Staubli VAL3: getFullError.pgx

public program getFullError(num x_nCamID (dimensions=1), num& x_nErrorCode (dimensions=1), string& x_sErrorMsg (dimensions=1))
  local num l_nErrorCode
begin
  //-----------------------------------------------------------------------
  //Header begin
  //Description of program
  //  Get error code of last executed command.
  //  Get error message from error message table (sMsgError).
  //
  //Input parameters
  //  num x_nCamID :
  //    role : camera's ID
  //
  //Output parameters
  //  string x_sMsgError :
  //    role : returns the error message
  //
  //  num x_nErrorCode:
  //    role : error code of the last executed command
  //
  //Examples
  //  call getFullError(l_nCamID,l_nError,l_sMsg)
  //
  //
  //History
  //  Creation : 17-04-12 - t.cail
  //
  //Header end
  //-----------------------------------------------------------------------
  //Read error code
  call getErrorCode(x_nCamID,x_nErrorCode)
  //Get corresponding error message
  call getErrorMessage(x_nErrorCode,x_sErrorMsg)
end
